(* PLC project Example1, KAIST_SELAB noNameNow 1.0 *)
(* stored: creationDateTime 2019-01-14T15:39:07, modificationDateTime 2019-02-19T14:16:39 *)

PROGRAM program0
  VAR
    R_TRIG_Switch : R_TRIG;
    SR_Manual : SR;
  END_VAR
  VAR_INPUT
    gDiSwitchManual : BOOL;
  END_VAR
  VAR_IN_OUT
    cmdManual : BOOL;
  END_VAR

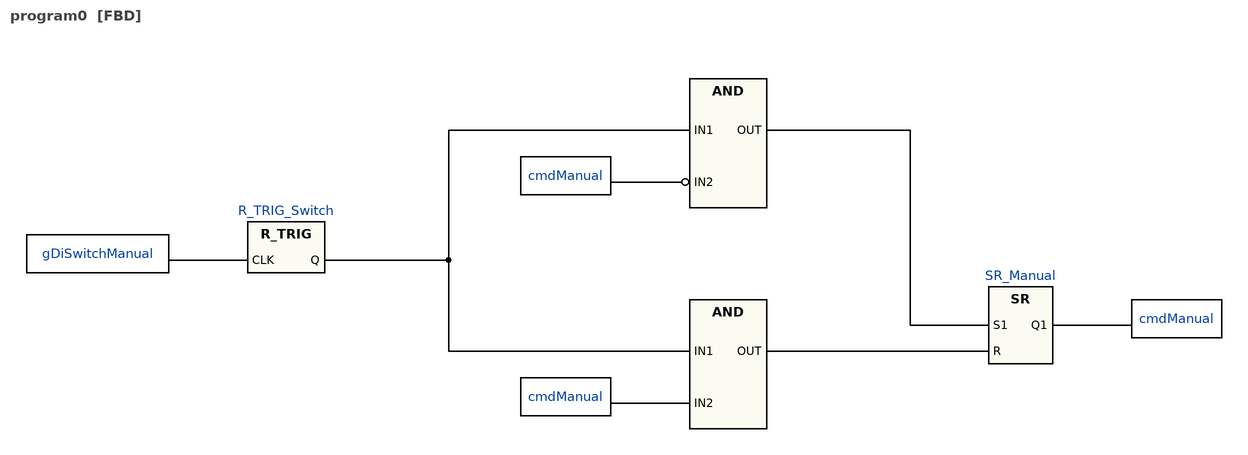
(* FBD diagram, written out as Structured Text *)
R_TRIG_Switch(CLK := gDiSwitchManual);
SR_Manual(S1 := R_TRIG_Switch.Q AND NOT cmdManual, R := R_TRIG_Switch.Q AND cmdManual);
cmdManual := SR_Manual.Q1;
END_PROGRAM
